// SIMATIC S7-200 project (STEP 7-Micro/WIN), CPU 221 REL 01.10

ORGANIZATION_BLOCK 主程序:OB1
TITLE=程序注释
BEGIN
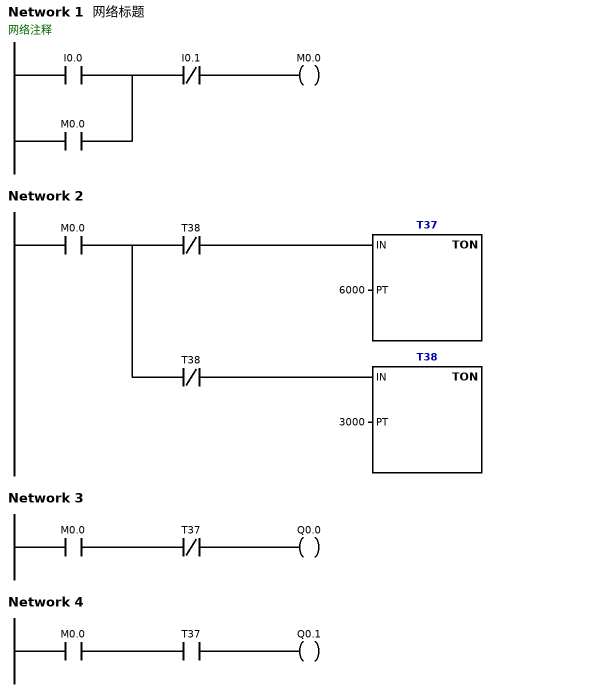
Network 1 // 网络标题
// 网络注释
LD     I0.0
O      M0.0
AN     I0.1
=      M0.0
Network 2
LD     M0.0
LPS
AN     T38
TON    T37, 6000
LPP
AN     T38
TON    T38, 3000
Network 3
LD     M0.0
AN     T37
=      Q0.0
Network 4
LD     M0.0
A      T37
=      Q0.1
END_ORGANIZATION_BLOCK
